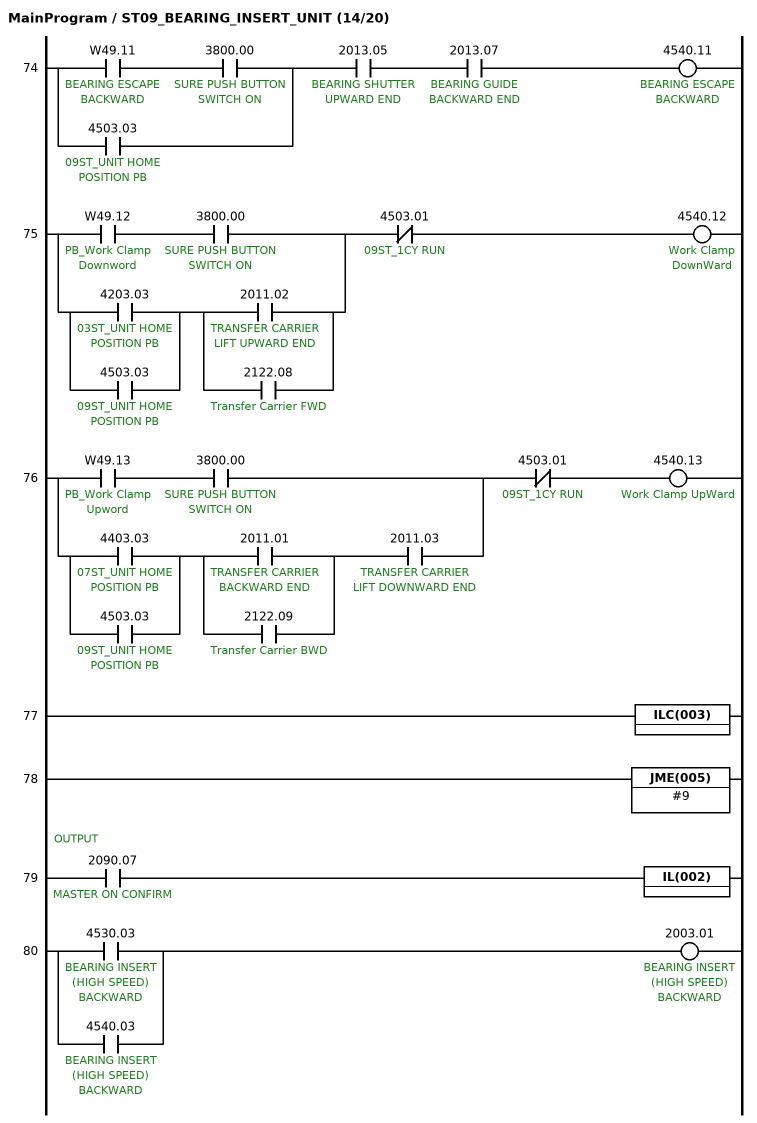
; [picture p480: MainProgram / ST09_BEARING_INSERT_UNIT, rungs 74-80]
; rung 74
LD W49.11  ; BEARING ESCAPE BACKWARD
AND 3800.00  ; SURE PUSH BUTTON SWITCH ON
OR 4503.03  ; 09ST_UNIT HOME POSITION PB
AND 2013.05  ; BEARING SHUTTER UPWARD END
AND 2013.07  ; BEARING GUIDE BACKWARD END
OUT 4540.11  ; BEARING ESCAPE BACKWARD
; rung 75
LD W49.12  ; PB_Work Clamp Downword
AND 3800.00  ; SURE PUSH BUTTON SWITCH ON
LD 4203.03  ; 03ST_UNIT HOME POSITION PB
OR 4503.03  ; 09ST_UNIT HOME POSITION PB
LD 2011.02  ; TRANSFER CARRIER LIFT UPWARD END
OR 2122.08  ; Transfer Carrier FWD
ANDLD
ORLD
ANDNOT 4503.01  ; 09ST_1CY RUN
OUT 4540.12  ; Work Clamp DownWard
; rung 76
LD W49.13  ; PB_Work Clamp Upword
AND 3800.00  ; SURE PUSH BUTTON SWITCH ON
LD 4403.03  ; 07ST_UNIT HOME POSITION PB
OR 4503.03  ; 09ST_UNIT HOME POSITION PB
LD 2011.01  ; TRANSFER CARRIER BACKWARD END
OR 2122.09  ; Transfer Carrier BWD
ANDLD
AND 2011.03  ; TRANSFER CARRIER LIFT DOWNWARD END
ORLD
ANDNOT 4503.01  ; 09ST_1CY RUN
OUT 4540.13  ; Work Clamp UpWard
; rung 77
ILC(003)
; rung 78
JME(005) #9
; rung 79: OUTPUT
LD 2090.07  ; MASTER ON CONFIRM
IL(002)
; rung 80
LD 4530.03  ; BEARING INSERT (HIGH SPEED) BACKWARD
OR 4540.03  ; BEARING INSERT (HIGH SPEED) BACKWARD
OUT 2003.01  ; BEARING INSERT (HIGH SPEED) BACKWARD

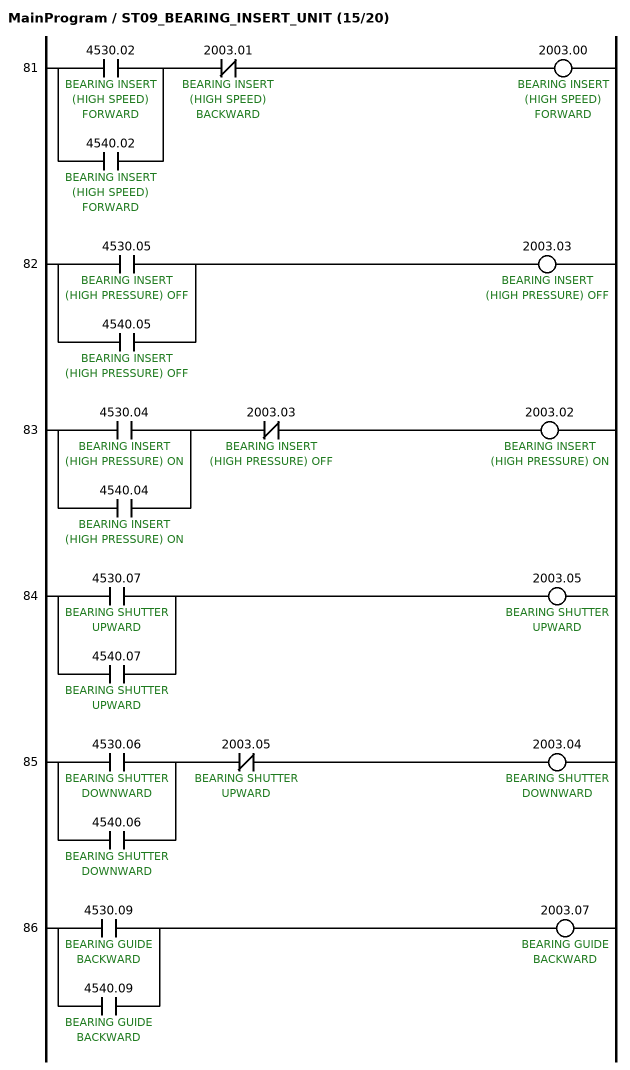
; rung 81
LD 4530.02  ; BEARING INSERT (HIGH SPEED) FORWARD
OR 4540.02  ; BEARING INSERT (HIGH SPEED) FORWARD
ANDNOT 2003.01  ; BEARING INSERT (HIGH SPEED) BACKWARD
OUT 2003.00  ; BEARING INSERT (HIGH SPEED) FORWARD
; rung 82
LD 4530.05  ; BEARING INSERT (HIGH PRESSURE) OFF
OR 4540.05  ; BEARING INSERT (HIGH PRESSURE) OFF
OUT 2003.03  ; BEARING INSERT (HIGH PRESSURE) OFF
; rung 83
LD 4530.04  ; BEARING INSERT (HIGH PRESSURE) ON
OR 4540.04  ; BEARING INSERT (HIGH PRESSURE) ON
ANDNOT 2003.03  ; BEARING INSERT (HIGH PRESSURE) OFF
OUT 2003.02  ; BEARING INSERT (HIGH PRESSURE) ON
; rung 84
LD 4530.07  ; BEARING SHUTTER UPWARD
OR 4540.07  ; BEARING SHUTTER UPWARD
OUT 2003.05  ; BEARING SHUTTER UPWARD
; rung 85
LD 4530.06  ; BEARING SHUTTER DOWNWARD
OR 4540.06  ; BEARING SHUTTER DOWNWARD
ANDNOT 2003.05  ; BEARING SHUTTER UPWARD
OUT 2003.04  ; BEARING SHUTTER DOWNWARD
; rung 86
LD 4530.09  ; BEARING GUIDE BACKWARD
OR 4540.09  ; BEARING GUIDE BACKWARD
OUT 2003.07  ; BEARING GUIDE BACKWARD

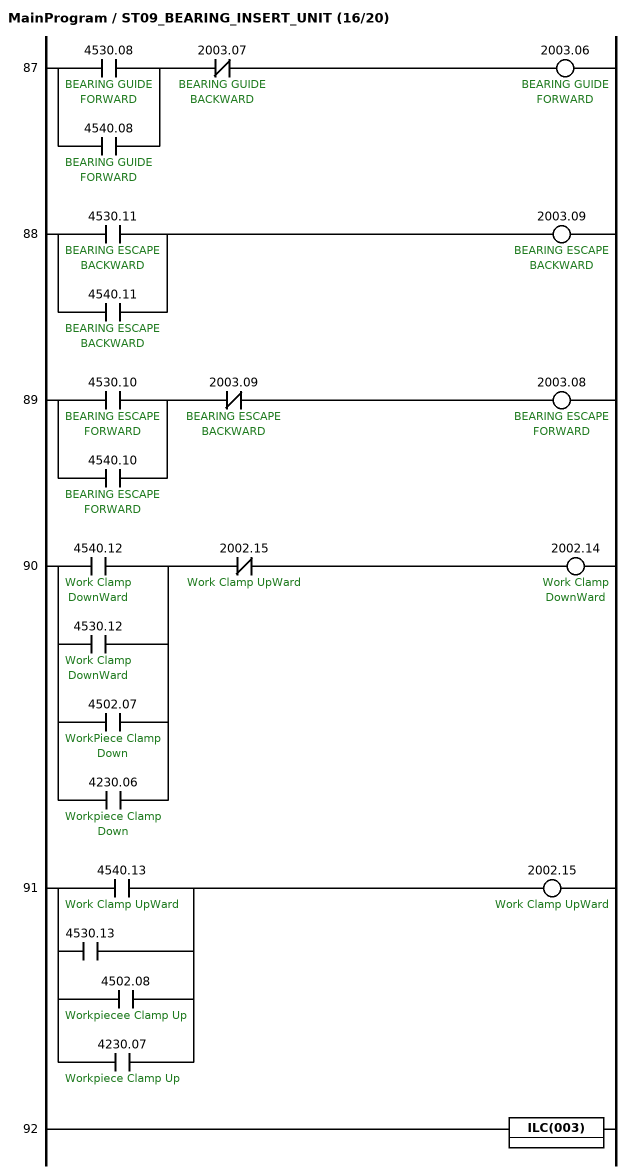
; rung 87
LD 4530.08  ; BEARING GUIDE FORWARD
OR 4540.08  ; BEARING GUIDE FORWARD
ANDNOT 2003.07  ; BEARING GUIDE BACKWARD
OUT 2003.06  ; BEARING GUIDE FORWARD
; rung 88
LD 4530.11  ; BEARING ESCAPE BACKWARD
OR 4540.11  ; BEARING ESCAPE BACKWARD
OUT 2003.09  ; BEARING ESCAPE BACKWARD
; rung 89
LD 4530.10  ; BEARING ESCAPE FORWARD
OR 4540.10  ; BEARING ESCAPE FORWARD
ANDNOT 2003.09  ; BEARING ESCAPE BACKWARD
OUT 2003.08  ; BEARING ESCAPE FORWARD
; rung 90
LD 4540.12  ; Work Clamp DownWard
OR 4530.12  ; Work Clamp DownWard
OR 4502.07  ; WorkPiece Clamp Down
OR 4230.06  ; Workpiece Clamp Down
ANDNOT 2002.15  ; Work Clamp UpWard
OUT 2002.14  ; Work Clamp DownWard
; rung 91
LD 4540.13  ; Work Clamp UpWard
OR 4530.13
OR 4502.08  ; Workpiecee Clamp Up
OR 4230.07  ; Workpiece Clamp Up
OUT 2002.15  ; Work Clamp UpWard
; rung 92
ILC(003)

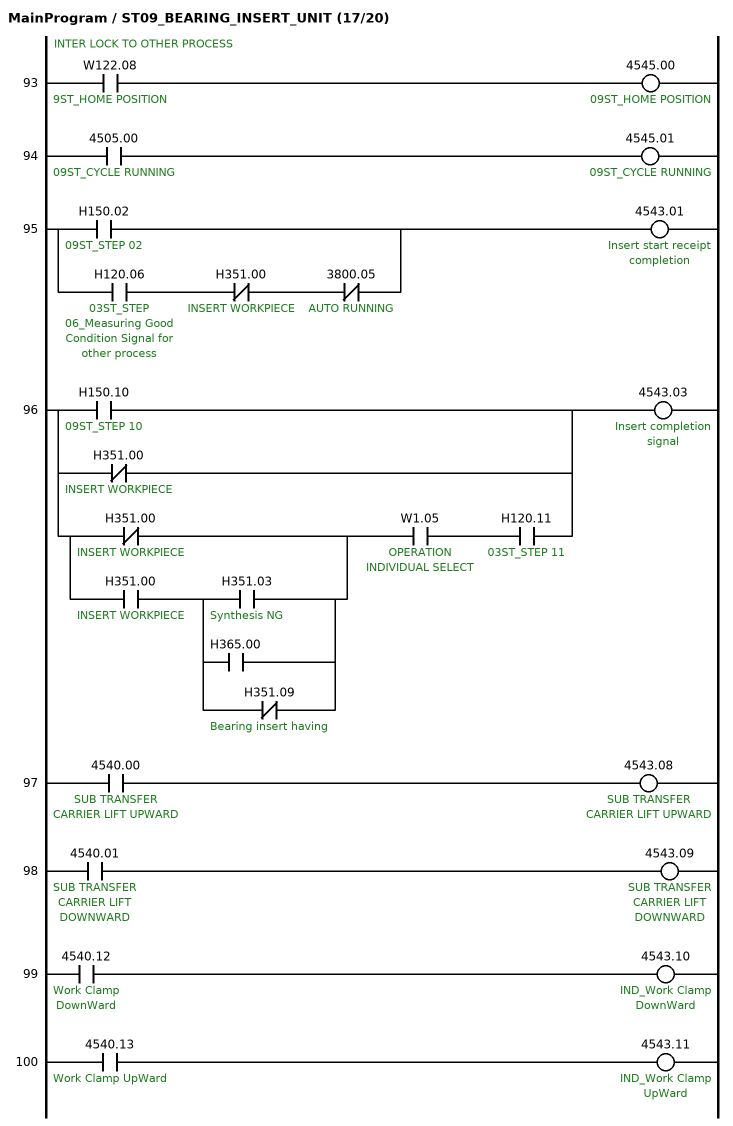
; rung 93: INTER LOCK TO OTHER PROCESS
LD W122.08  ; 9ST_HOME POSITION
OUT 4545.00  ; 09ST_HOME POSITION
; rung 94
LD 4505.00  ; 09ST_CYCLE RUNNING
OUT 4545.01  ; 09ST_CYCLE RUNNING
; rung 95
LD H150.02  ; 09ST_STEP 02
LD H120.06  ; 03ST_STEP 06_Measuring Good Condition Signal for other process
ANDNOT H351.00  ; INSERT WORKPIECE
ANDNOT 3800.05  ; AUTO RUNNING
ORLD
OUT 4543.01  ; Insert start receipt completion
; rung 96
LD H150.10  ; 09ST_STEP 10
ORNOT H351.00  ; INSERT WORKPIECE
LDNOT H351.00  ; INSERT WORKPIECE
LD H351.00  ; INSERT WORKPIECE
LD H351.03  ; Synthesis NG
OR H365.00
ORNOT H351.09  ; Bearing insert having
ANDLD
ORLD
AND W1.05  ; OPERATION INDIVIDUAL SELECT
AND H120.11  ; 03ST_STEP 11
ORLD
OUT 4543.03  ; Insert completion signal
; rung 97
LD 4540.00  ; SUB TRANSFER CARRIER LIFT UPWARD
OUT 4543.08  ; SUB TRANSFER CARRIER LIFT UPWARD
; rung 98
LD 4540.01  ; SUB TRANSFER CARRIER LIFT DOWNWARD
OUT 4543.09  ; SUB TRANSFER CARRIER LIFT DOWNWARD
; rung 99
LD 4540.12  ; Work Clamp DownWard
OUT 4543.10  ; IND_Work Clamp DownWard
; rung 100
LD 4540.13  ; Work Clamp UpWard
OUT 4543.11  ; IND_Work Clamp UpWard

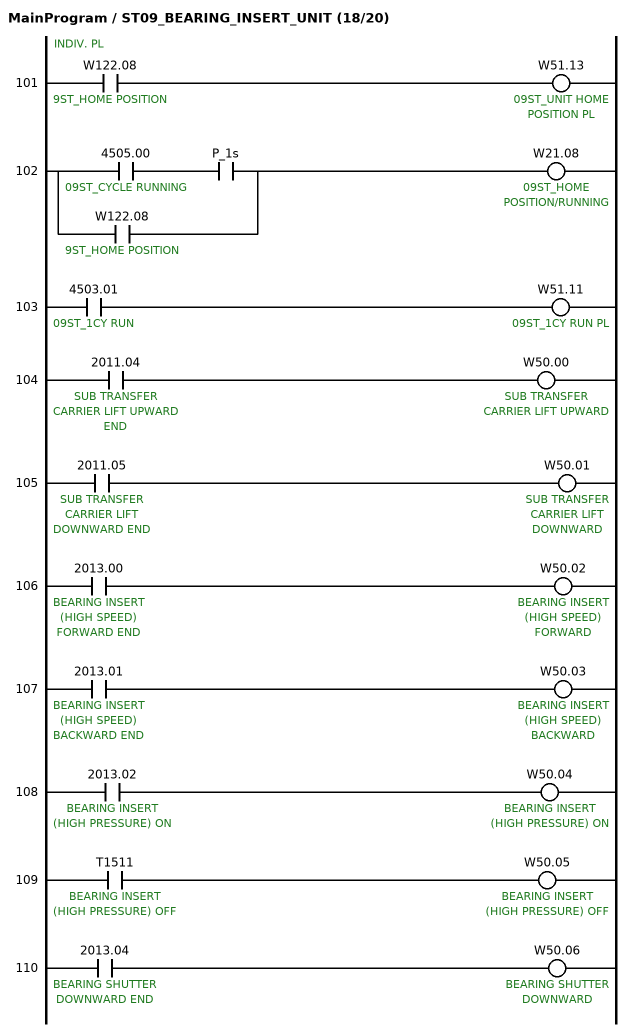
; rung 101: INDIV. PL
LD W122.08  ; 9ST_HOME POSITION
OUT W51.13  ; 09ST_UNIT HOME POSITION PL
; rung 102
LD 4505.00  ; 09ST_CYCLE RUNNING
AND P_1s
OR W122.08  ; 9ST_HOME POSITION
OUT W21.08  ; 09ST_HOME POSITION/RUNNING
; rung 103
LD 4503.01  ; 09ST_1CY RUN
OUT W51.11  ; 09ST_1CY RUN PL
; rung 104
LD 2011.04  ; SUB TRANSFER CARRIER LIFT UPWARD END
OUT W50.00  ; SUB TRANSFER CARRIER LIFT UPWARD
; rung 105
LD 2011.05  ; SUB TRANSFER CARRIER LIFT DOWNWARD END
OUT W50.01  ; SUB TRANSFER CARRIER LIFT DOWNWARD
; rung 106
LD 2013.00  ; BEARING INSERT (HIGH SPEED) FORWARD END
OUT W50.02  ; BEARING INSERT (HIGH SPEED) FORWARD
; rung 107
LD 2013.01  ; BEARING INSERT (HIGH SPEED) BACKWARD END
OUT W50.03  ; BEARING INSERT (HIGH SPEED) BACKWARD
; rung 108
LD 2013.02  ; BEARING INSERT (HIGH PRESSURE) ON
OUT W50.04  ; BEARING INSERT (HIGH PRESSURE) ON
; rung 109
LD T1511  ; BEARING INSERT (HIGH PRESSURE) OFF
OUT W50.05  ; BEARING INSERT (HIGH PRESSURE) OFF
; rung 110
LD 2013.04  ; BEARING SHUTTER DOWNWARD END
OUT W50.06  ; BEARING SHUTTER DOWNWARD

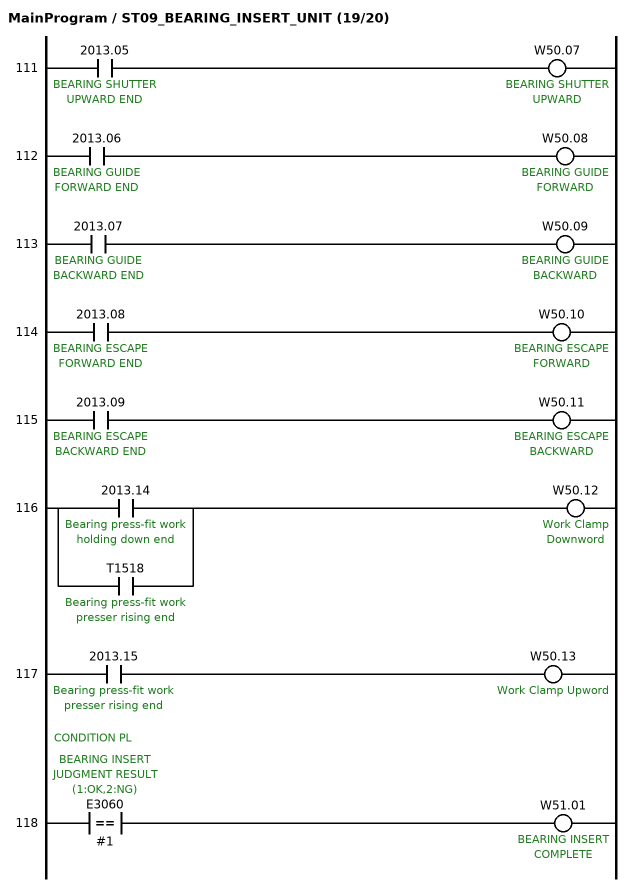
; rung 111
LD 2013.05  ; BEARING SHUTTER UPWARD END
OUT W50.07  ; BEARING SHUTTER UPWARD
; rung 112
LD 2013.06  ; BEARING GUIDE FORWARD END
OUT W50.08  ; BEARING GUIDE FORWARD
; rung 113
LD 2013.07  ; BEARING GUIDE BACKWARD END
OUT W50.09  ; BEARING GUIDE BACKWARD
; rung 114
LD 2013.08  ; BEARING ESCAPE FORWARD END
OUT W50.10  ; BEARING ESCAPE FORWARD
; rung 115
LD 2013.09  ; BEARING ESCAPE BACKWARD END
OUT W50.11  ; BEARING ESCAPE BACKWARD
; rung 116
LD 2013.14  ; Bearing press-fit work holding down end
OR T1518  ; Bearing press-fit work presser rising end
OUT W50.12  ; Work Clamp Downword
; rung 117
LD 2013.15  ; Bearing press-fit work presser rising end
OUT W50.13  ; Work Clamp Upword
; rung 118: CONDITION PL
LD=(300) E3060 #1  ; BEARING INSERT JUDGMENT RESULT (1:OK,2:NG)
OUT W51.01  ; BEARING INSERT COMPLETE

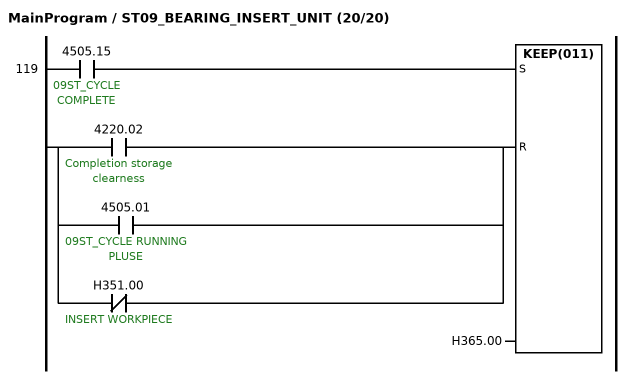
; rung 119
LD 4505.15  ; 09ST_CYCLE COMPLETE
LD 4220.02  ; Completion storage clearness
OR 4505.01  ; 09ST_CYCLE RUNNING PLUSE
ORNOT H351.00  ; INSERT WORKPIECE
KEEP(011) H365.00

### Section ST10_LENGTH_MEASURE_UNIT

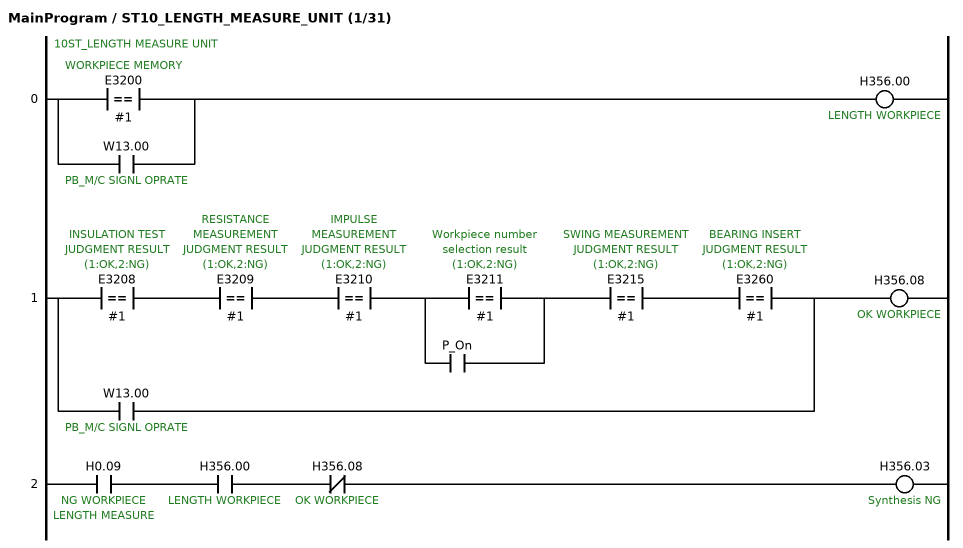
; rung 0: 10ST_LENGTH MEASURE UNIT
LD=(300) E3200 #1  ; WORKPIECE MEMORY
OR W13.00  ; PB_M/C SIGNL OPRATE
OUT H356.00  ; LENGTH WORKPIECE
; rung 1
LD=(300) E3208 #1  ; INSULATION TEST JUDGMENT RESULT (1:OK,2:NG)
AND=(300) E3209 #1  ; RESISTANCE MEASUREMENT JUDGMENT RESULT (1:OK,2:NG)
AND=(300) E3210 #1  ; IMPULSE MEASUREMENT JUDGMENT RESULT (1:OK,2:NG)
LD=(300) E3211 #1  ; Workpiece number selection result (1:OK,2:NG)
OR P_On
ANDLD
AND=(300) E3215 #1  ; SWING MEASUREMENT JUDGMENT RESULT (1:OK,2:NG)
AND=(300) E3260 #1  ; BEARING INSERT JUDGMENT RESULT (1:OK,2:NG)
OR W13.00  ; PB_M/C SIGNL OPRATE
OUT H356.08  ; OK WORKPIECE
; rung 2
LD H0.09  ; NG WORKPIECE LENGTH MEASURE
AND H356.00  ; LENGTH WORKPIECE
ANDNOT H356.08  ; OK WORKPIECE
OUT H356.03  ; Synthesis NG

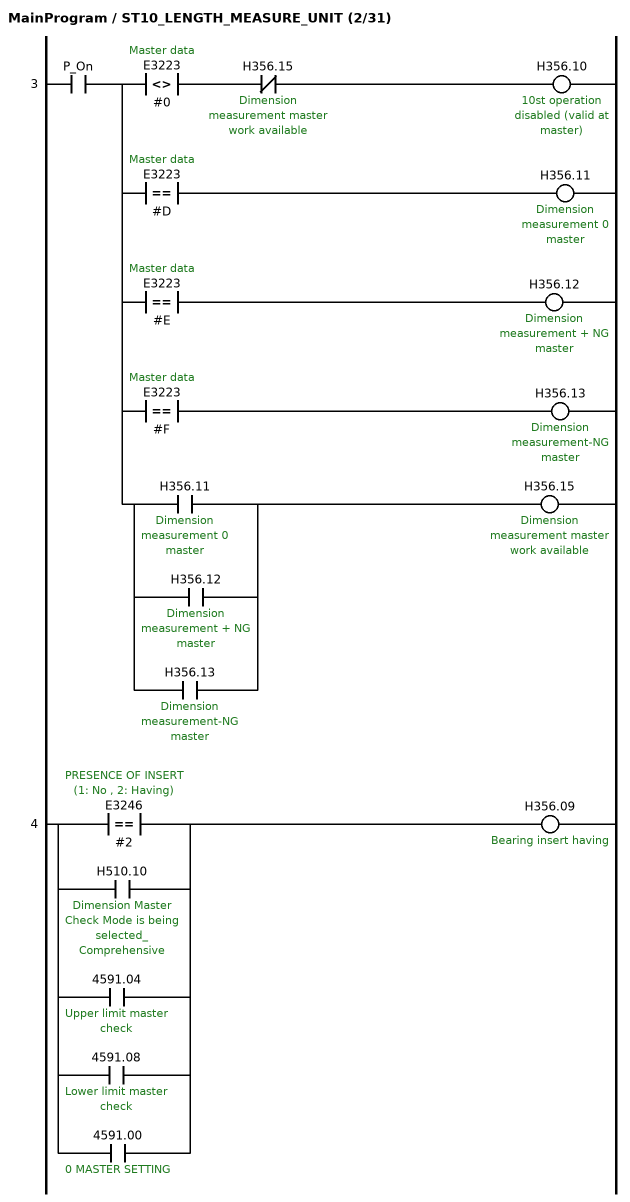
; rung 3
LD P_On
OUT TR0
AND<>(305) E3223 #0  ; Master data
ANDNOT H356.15  ; Dimension measurement master work available
OUT H356.10  ; 10st operation disabled (valid at master)
LD TR0
AND=(300) E3223 #D  ; Master data
OUT H356.11  ; Dimension measurement 0 master
LD TR0
AND=(300) E3223 #E  ; Master data
OUT H356.12  ; Dimension measurement + NG master
LD TR0
AND=(300) E3223 #F  ; Master data
OUT H356.13  ; Dimension measurement-NG master
LD TR0
LD H356.11  ; Dimension measurement 0 master
OR H356.12  ; Dimension measurement + NG master
OR H356.13  ; Dimension measurement-NG master
ANDLD
OUT H356.15  ; Dimension measurement master work available
; rung 4
LD=(300) E3246 #2  ; PRESENCE OF INSERT (1: No , 2: Having)
OR H510.10  ; Dimension Master Check Mode is being selected_Comprehensive
OR 4591.04  ; Upper limit master check
OR 4591.08  ; Lower limit master check
OR 4591.00  ; 0 MASTER SETTING
OUT H356.09  ; Bearing insert having

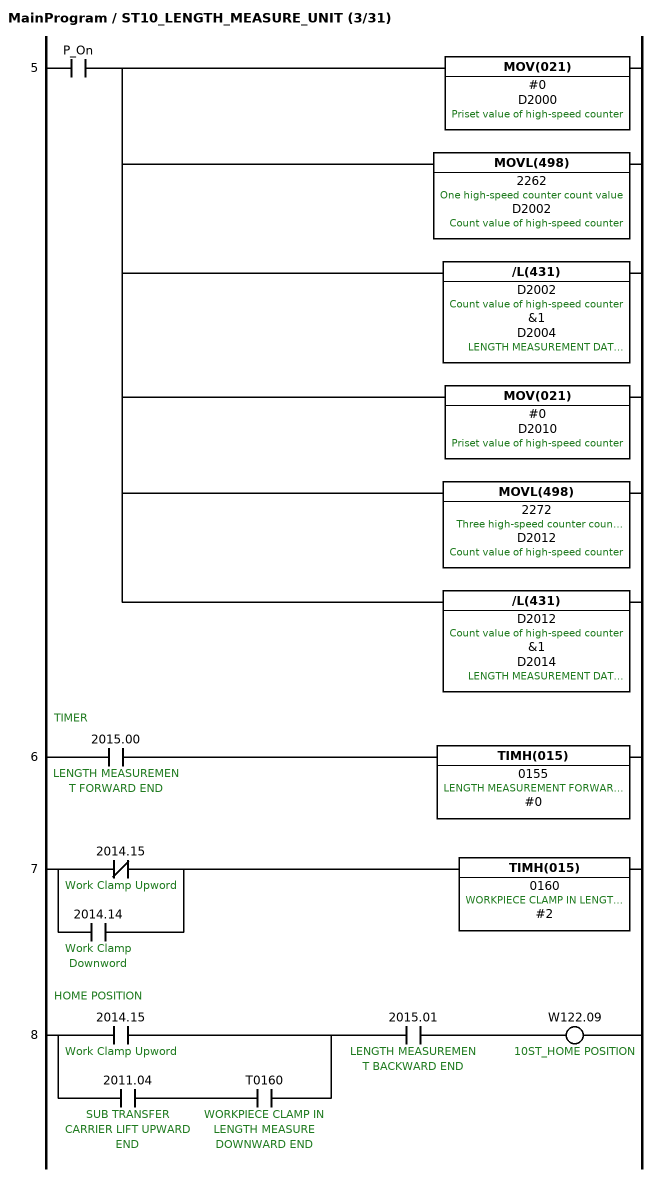
; rung 5
LD P_On
MOV(021) #0 D2000  ; Priset value of high-speed counter
MOVL(498) 2262 D2002  ; One high-speed counter count value, Count value of high-speed counter
/L(431) D2002 &1 D2004  ; Count value of high-speed counter, LENGTH MEASUREMENT DATA (OVERALL)
MOV(021) #0 D2010  ; Priset value of high-speed counter
MOVL(498) 2272 D2012  ; Three high-speed counter count value, Count value of high-speed counter
/L(431) D2012 &1 D2014  ; Count value of high-speed counter, LENGTH MEASUREMENT DATA (BEARING)
; rung 6: TIMER
LD 2015.00  ; LENGTH MEASUREMENT FORWARD END
TIMH(015) 0155 #0  ; LENGTH MEASUREMENT FORWARD END
; rung 7
LDNOT 2014.15  ; Work Clamp Upword
OR 2014.14  ; Work Clamp Downword
TIMH(015) 0160 #2  ; WORKPIECE CLAMP IN LENGTH MEASURE DOWNWARD END
; rung 8: HOME POSITION
LD 2014.15  ; Work Clamp Upword
LD 2011.04  ; SUB TRANSFER CARRIER LIFT UPWARD END
AND T0160  ; WORKPIECE CLAMP IN LENGTH MEASURE DOWNWARD END
ORLD
AND 2015.01  ; LENGTH MEASUREMENT BACKWARD END
OUT W122.09  ; 10ST_HOME POSITION

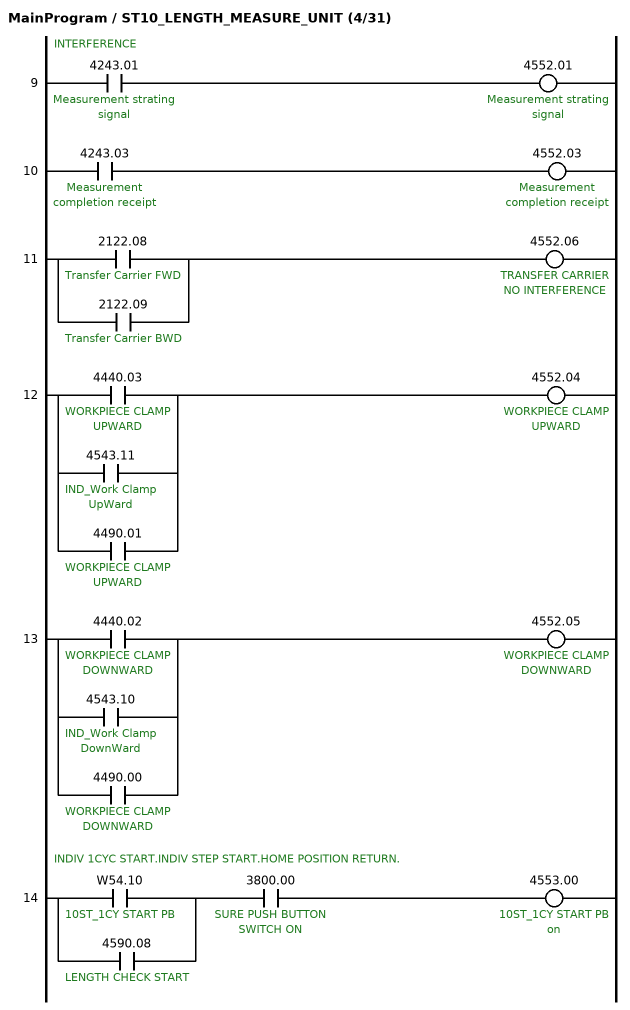
; rung 9: INTERFERENCE
LD 4243.01  ; Measurement strating signal
OUT 4552.01  ; Measurement strating signal
; rung 10
LD 4243.03  ; Measurement completion receipt
OUT 4552.03  ; Measurement completion receipt
; rung 11
LD 2122.08  ; Transfer Carrier FWD
OR 2122.09  ; Transfer Carrier BWD
OUT 4552.06  ; TRANSFER CARRIER NO INTERFERENCE
; rung 12
LD 4440.03  ; WORKPIECE CLAMP UPWARD
OR 4543.11  ; IND_Work Clamp UpWard
OR 4490.01  ; WORKPIECE CLAMP UPWARD
OUT 4552.04  ; WORKPIECE CLAMP UPWARD
; rung 13
LD 4440.02  ; WORKPIECE CLAMP DOWNWARD
OR 4543.10  ; IND_Work Clamp DownWard
OR 4490.00  ; WORKPIECE CLAMP DOWNWARD
OUT 4552.05  ; WORKPIECE CLAMP DOWNWARD
; rung 14: INDIV 1CYC START.INDIV STEP START.HOME POSITION RETURN.
LD W54.10  ; 10ST_1CY START PB
OR 4590.08  ; LENGTH CHECK START
AND 3800.00  ; SURE PUSH BUTTON SWITCH ON
OUT 4553.00  ; 10ST_1CY START PB on

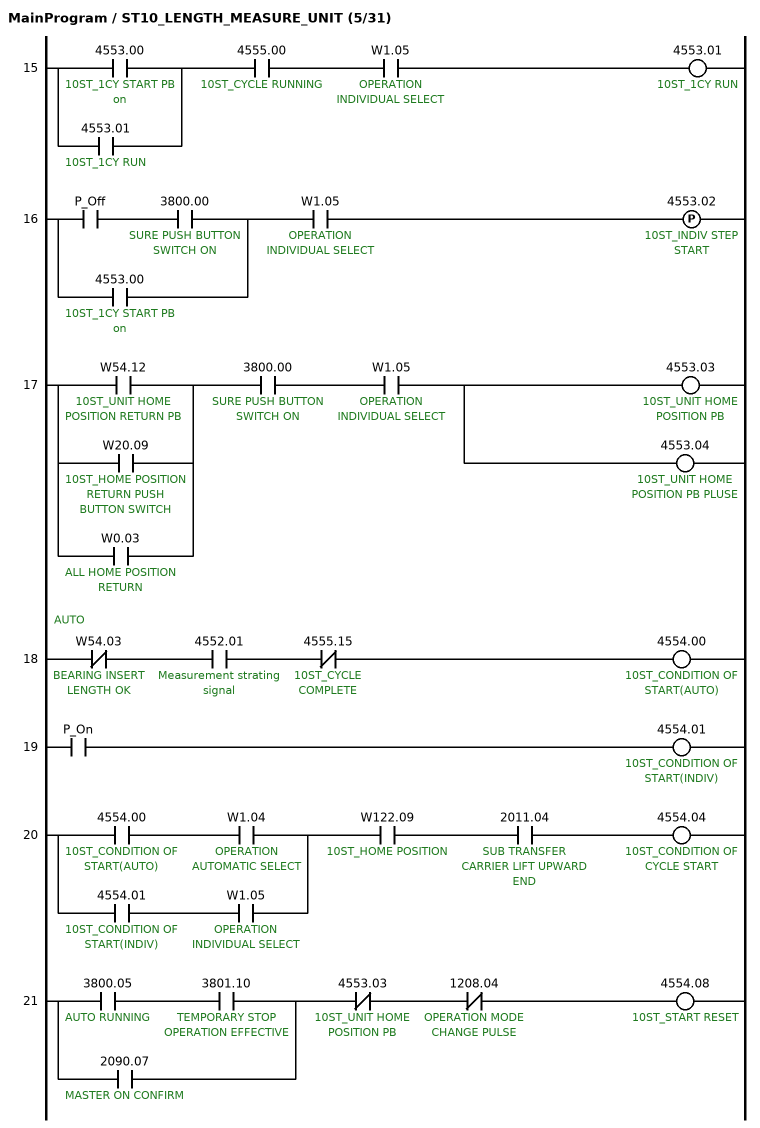
; rung 15
LD 4553.00  ; 10ST_1CY START PB on
OR 4553.01  ; 10ST_1CY RUN
AND 4555.00  ; 10ST_CYCLE RUNNING
AND W1.05  ; OPERATION INDIVIDUAL SELECT
OUT 4553.01  ; 10ST_1CY RUN
; rung 16
LD P_Off
AND 3800.00  ; SURE PUSH BUTTON SWITCH ON
OR 4553.00  ; 10ST_1CY START PB on
AND W1.05  ; OPERATION INDIVIDUAL SELECT
DIFU(013) 4553.02  ; 10ST_INDIV STEP START
; rung 17
LD W54.12  ; 10ST_UNIT HOME POSITION RETURN PB
OR W20.09  ; 10ST_HOME POSITION RETURN PUSH BUTTON SWITCH
OR W0.03  ; ALL HOME POSITION RETURN
AND 3800.00  ; SURE PUSH BUTTON SWITCH ON
AND W1.05  ; OPERATION INDIVIDUAL SELECT
OUT 4553.03  ; 10ST_UNIT HOME POSITION PB
OUT 4553.04  ; 10ST_UNIT HOME POSITION PB PLUSE
; rung 18: AUTO
LDNOT W54.03  ; BEARING INSERT LENGTH OK
AND 4552.01  ; Measurement strating signal
ANDNOT 4555.15  ; 10ST_CYCLE COMPLETE
OUT 4554.00  ; 10ST_CONDITION OF START(AUTO)
; rung 19
LD P_On
OUT 4554.01  ; 10ST_CONDITION OF START(INDIV)
; rung 20
LD 4554.00  ; 10ST_CONDITION OF START(AUTO)
AND W1.04  ; OPERATION AUTOMATIC SELECT
LD 4554.01  ; 10ST_CONDITION OF START(INDIV)
AND W1.05  ; OPERATION INDIVIDUAL SELECT
ORLD
AND W122.09  ; 10ST_HOME POSITION
AND 2011.04  ; SUB TRANSFER CARRIER LIFT UPWARD END
OUT 4554.04  ; 10ST_CONDITION OF CYCLE START
; rung 21
LD 3800.05  ; AUTO RUNNING
AND 3801.10  ; TEMPORARY STOP OPERATION EFFECTIVE
OR 2090.07  ; MASTER ON CONFIRM
ANDNOT 4553.03  ; 10ST_UNIT HOME POSITION PB
ANDNOT 1208.04  ; OPERATION MODE CHANGE PULSE
OUT 4554.08  ; 10ST_START RESET

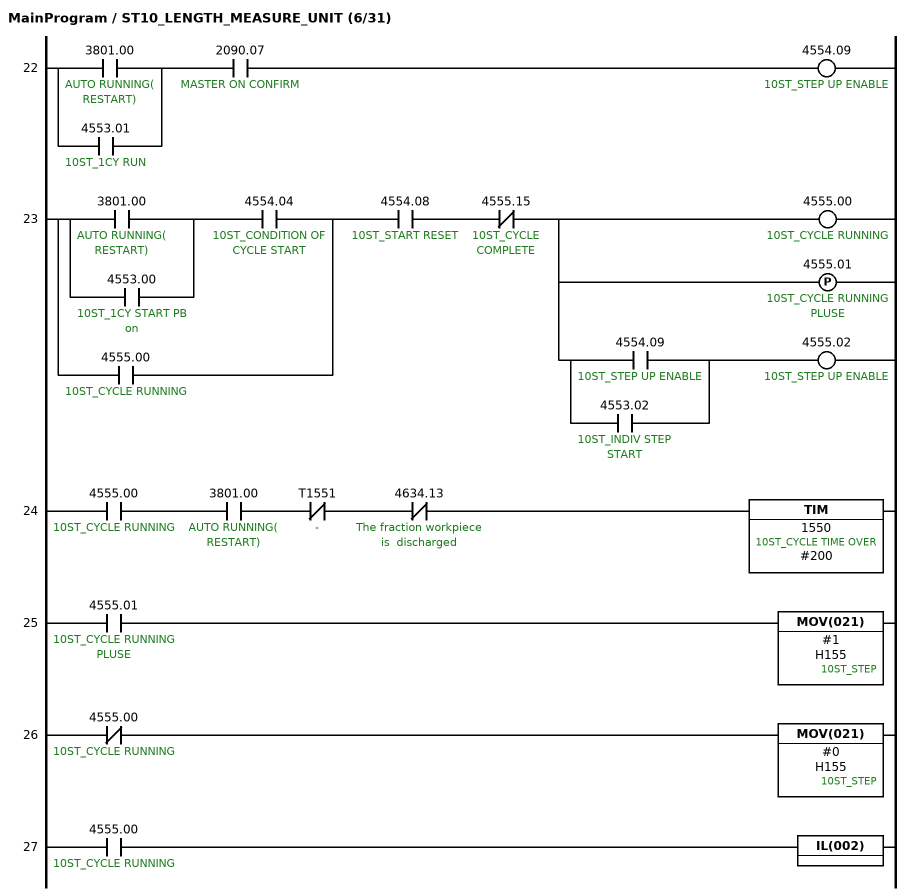
; rung 22
LD 3801.00  ; AUTO RUNNING(RESTART)
OR 4553.01  ; 10ST_1CY RUN
AND 2090.07  ; MASTER ON CONFIRM
OUT 4554.09  ; 10ST_STEP UP ENABLE
; rung 23
LD 3801.00  ; AUTO RUNNING(RESTART)
OR 4553.00  ; 10ST_1CY START PB on
AND 4554.04  ; 10ST_CONDITION OF CYCLE START
OR 4555.00  ; 10ST_CYCLE RUNNING
AND 4554.08  ; 10ST_START RESET
ANDNOT 4555.15  ; 10ST_CYCLE COMPLETE
OUT 4555.00  ; 10ST_CYCLE RUNNING
DIFU(013) 4555.01  ; 10ST_CYCLE RUNNING PLUSE
LD 4554.09  ; 10ST_STEP UP ENABLE
OR 4553.02  ; 10ST_INDIV STEP START
ANDLD
OUT 4555.02  ; 10ST_STEP UP ENABLE
; rung 24
LD 4555.00  ; 10ST_CYCLE RUNNING
AND 3801.00  ; AUTO RUNNING(RESTART)
ANDNOT T1551  ; -
ANDNOT 4634.13  ; The fraction workpiece is  discharged
TIM 1550 #200  ; 10ST_CYCLE TIME OVER
; rung 25
LD 4555.01  ; 10ST_CYCLE RUNNING PLUSE
MOV(021) #1 H155  ; 10ST_STEP
; rung 26
LDNOT 4555.00  ; 10ST_CYCLE RUNNING
MOV(021) #0 H155  ; 10ST_STEP
; rung 27
LD 4555.00  ; 10ST_CYCLE RUNNING
IL(002)

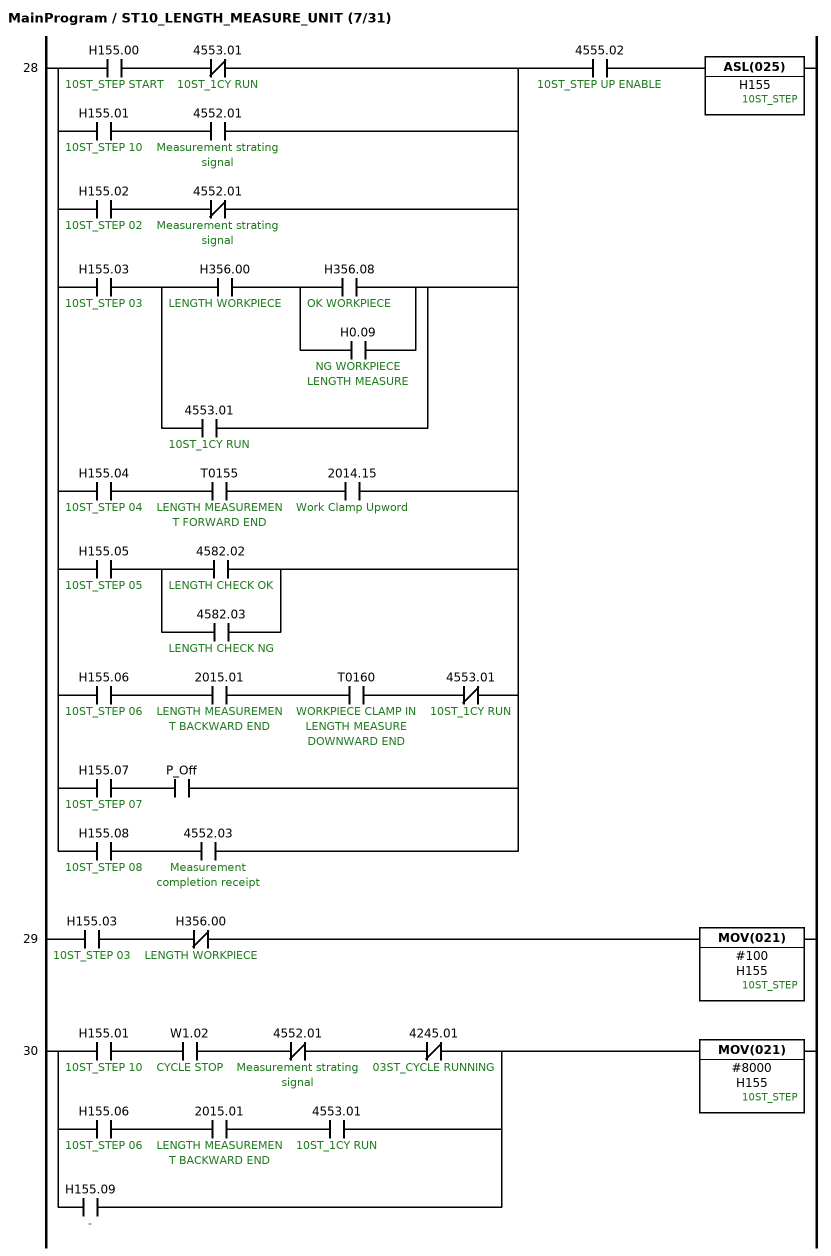
; rung 28
LD H155.00  ; 10ST_STEP START
ANDNOT 4553.01  ; 10ST_1CY RUN
LD H155.01  ; 10ST_STEP 10
AND 4552.01  ; Measurement strating signal
ORLD
LD H155.02  ; 10ST_STEP 02
ANDNOT 4552.01  ; Measurement strating signal
ORLD
LD H155.03  ; 10ST_STEP 03
LD H356.00  ; LENGTH WORKPIECE
LD H356.08  ; OK WORKPIECE
OR H0.09  ; NG WORKPIECE LENGTH MEASURE
ANDLD
OR 4553.01  ; 10ST_1CY RUN
ANDLD
ORLD
LD H155.04  ; 10ST_STEP 04
AND T0155  ; LENGTH MEASUREMENT FORWARD END
AND 2014.15  ; Work Clamp Upword
ORLD
LD H155.05  ; 10ST_STEP 05
LD 4582.02  ; LENGTH CHECK OK
OR 4582.03  ; LENGTH CHECK NG
ANDLD
ORLD
LD H155.06  ; 10ST_STEP 06
AND 2015.01  ; LENGTH MEASUREMENT BACKWARD END
AND T0160  ; WORKPIECE CLAMP IN LENGTH MEASURE DOWNWARD END
ANDNOT 4553.01  ; 10ST_1CY RUN
ORLD
LD H155.07  ; 10ST_STEP 07
AND P_Off
ORLD
LD H155.08  ; 10ST_STEP 08
AND 4552.03  ; Measurement completion receipt
ORLD
AND 4555.02  ; 10ST_STEP UP ENABLE
ASL(025) H155  ; 10ST_STEP
; rung 29
LD H155.03  ; 10ST_STEP 03
ANDNOT H356.00  ; LENGTH WORKPIECE
MOV(021) #100 H155  ; 10ST_STEP
; rung 30
LD H155.01  ; 10ST_STEP 10
AND W1.02  ; CYCLE STOP
ANDNOT 4552.01  ; Measurement strating signal
ANDNOT 4245.01  ; 03ST_CYCLE RUNNING
LD H155.06  ; 10ST_STEP 06
AND 2015.01  ; LENGTH MEASUREMENT BACKWARD END
AND 4553.01  ; 10ST_1CY RUN
ORLD
OR H155.09  ; -
MOV(021) #8000 H155  ; 10ST_STEP

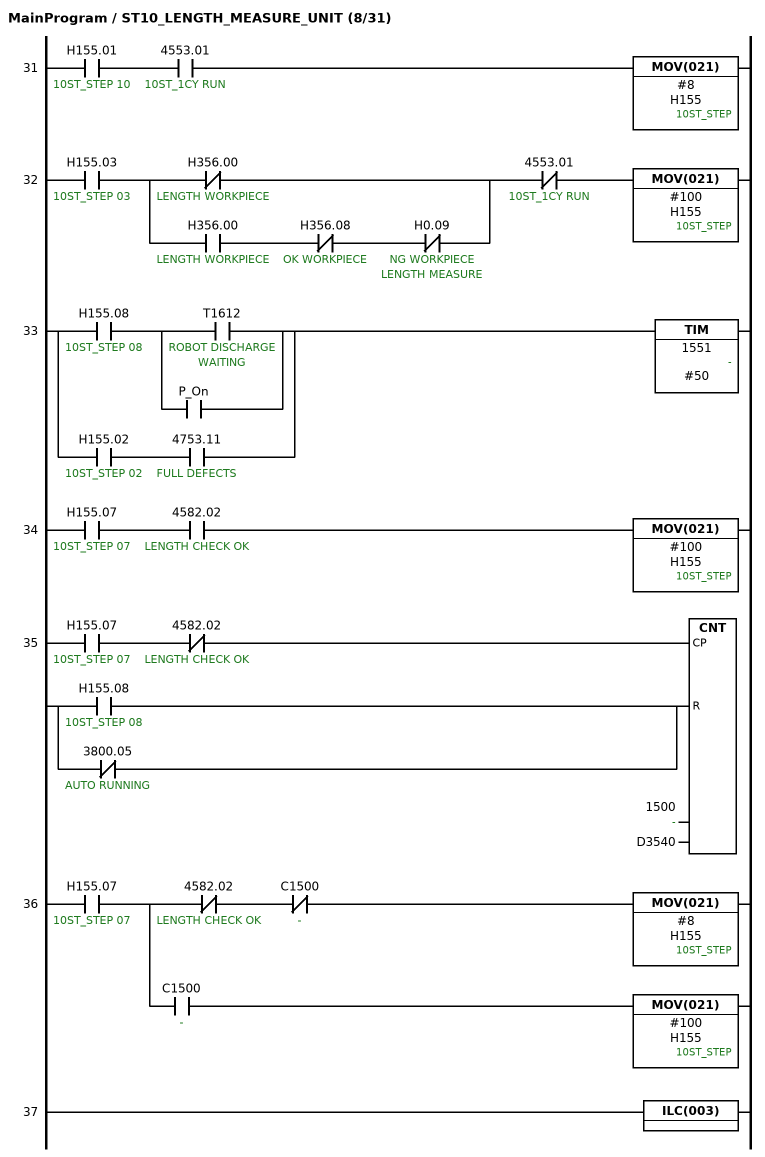
; rung 31
LD H155.01  ; 10ST_STEP 10
AND 4553.01  ; 10ST_1CY RUN
MOV(021) #8 H155  ; 10ST_STEP
; rung 32
LD H155.03  ; 10ST_STEP 03
LDNOT H356.00  ; LENGTH WORKPIECE
LD H356.00  ; LENGTH WORKPIECE
ANDNOT H356.08  ; OK WORKPIECE
ANDNOT H0.09  ; NG WORKPIECE LENGTH MEASURE
ORLD
ANDLD
ANDNOT 4553.01  ; 10ST_1CY RUN
MOV(021) #100 H155  ; 10ST_STEP
; rung 33
LD H155.08  ; 10ST_STEP 08
LD T1612  ; ROBOT DISCHARGE WAITING
OR P_On
ANDLD
LD H155.02  ; 10ST_STEP 02
AND 4753.11  ; FULL DEFECTS
ORLD
TIM 1551 #50  ; -
; rung 34
LD H155.07  ; 10ST_STEP 07
AND 4582.02  ; LENGTH CHECK OK
MOV(021) #100 H155  ; 10ST_STEP
; rung 35
LD H155.07  ; 10ST_STEP 07
ANDNOT 4582.02  ; LENGTH CHECK OK
LD H155.08  ; 10ST_STEP 08
ORNOT 3800.05  ; AUTO RUNNING
CNT 1500 D3540  ; -
; rung 36
LD H155.07  ; 10ST_STEP 07
OUT TR0
ANDNOT 4582.02  ; LENGTH CHECK OK
ANDNOT C1500  ; -
MOV(021) #8 H155  ; 10ST_STEP
LD TR0
AND C1500  ; -
MOV(021) #100 H155  ; 10ST_STEP
; rung 37
ILC(003)

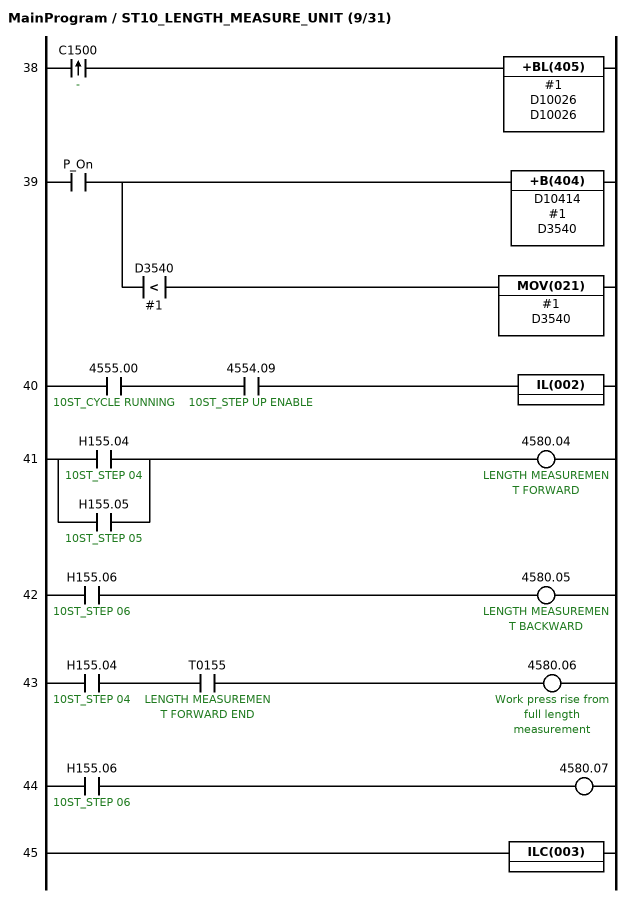
; rung 38
@LD C1500  ; -
+BL(405) #1 D10026 D10026
; rung 39
LD P_On
+B(404) D10414 #1 D3540
AND<(310) D3540 #1
MOV(021) #1 D3540
; rung 40
LD 4555.00  ; 10ST_CYCLE RUNNING
AND 4554.09  ; 10ST_STEP UP ENABLE
IL(002)
; rung 41
LD H155.04  ; 10ST_STEP 04
OR H155.05  ; 10ST_STEP 05
OUT 4580.04  ; LENGTH MEASUREMENT FORWARD
; rung 42
LD H155.06  ; 10ST_STEP 06
OUT 4580.05  ; LENGTH MEASUREMENT BACKWARD
; rung 43
LD H155.04  ; 10ST_STEP 04
AND T0155  ; LENGTH MEASUREMENT FORWARD END
OUT 4580.06  ; Work press rise from full length measurement
; rung 44
LD H155.06  ; 10ST_STEP 06
OUT 4580.07
; rung 45
ILC(003)

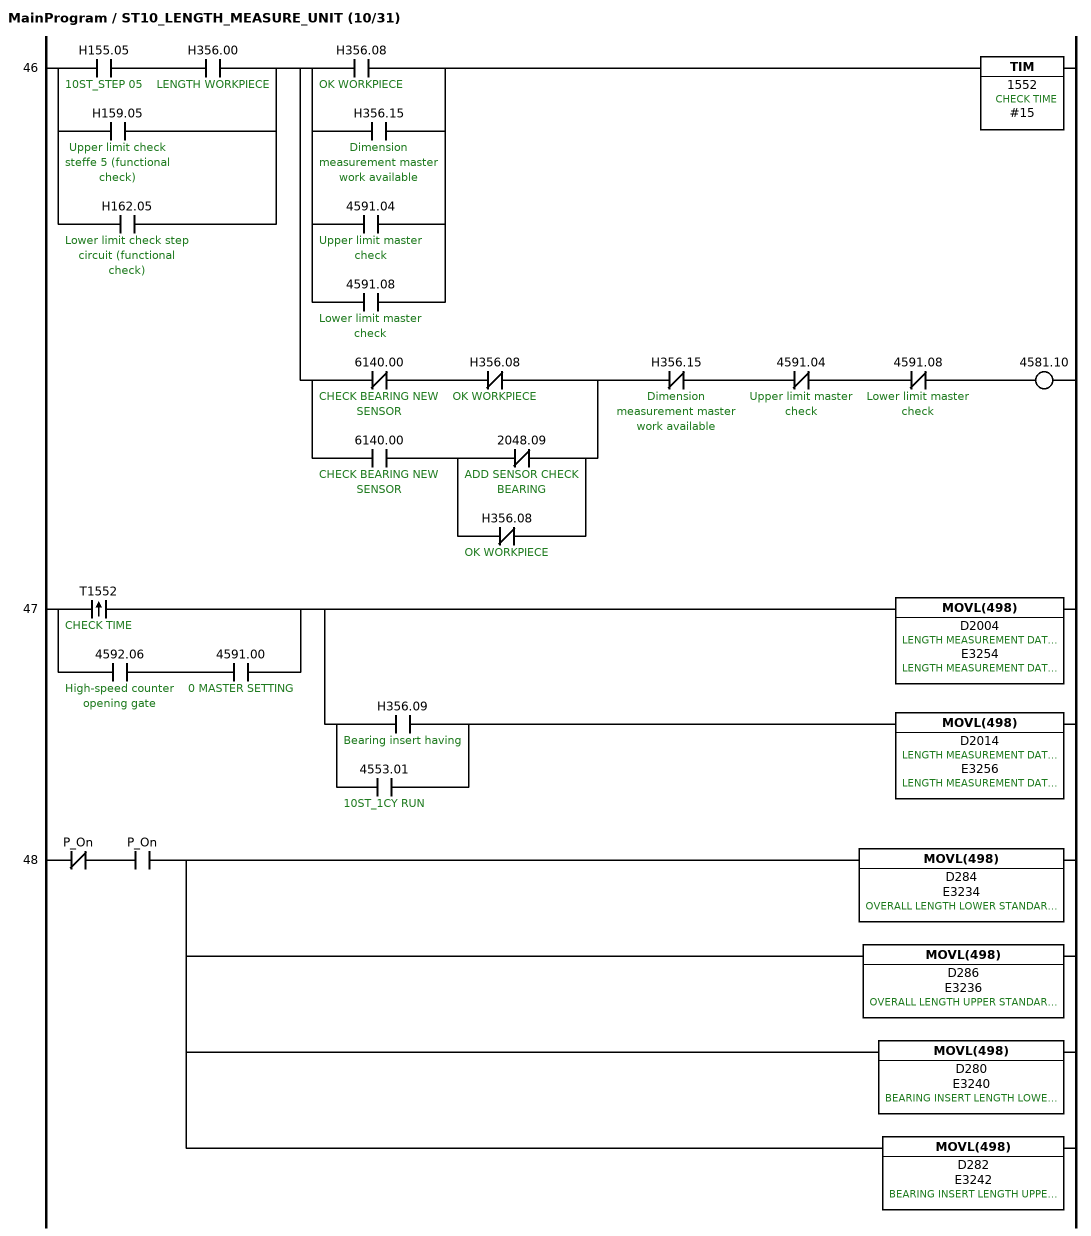
; rung 46
LD H155.05  ; 10ST_STEP 05
AND H356.00  ; LENGTH WORKPIECE
OR H159.05  ; Upper limit check steffe 5 (functional check)
OR H162.05  ; Lower limit check step circuit (functional check)
OUT TR0
LD H356.08  ; OK WORKPIECE
OR H356.15  ; Dimension measurement master work available
OR 4591.04  ; Upper limit master check
OR 4591.08  ; Lower limit master check
ANDLD
TIM 1552 #15  ; CHECK TIME
LD TR0
LDNOT 6140.00  ; CHECK BEARING NEW SENSOR
ANDNOT H356.08  ; OK WORKPIECE
LD 6140.00  ; CHECK BEARING NEW SENSOR
LDNOT 2048.09  ; ADD SENSOR CHECK BEARING
ORNOT H356.08  ; OK WORKPIECE
ANDLD
ORLD
ANDLD
ANDNOT H356.15  ; Dimension measurement master work available
ANDNOT 4591.04  ; Upper limit master check
ANDNOT 4591.08  ; Lower limit master check
OUT 4581.10
; rung 47
@LD T1552  ; CHECK TIME
LD 4592.06  ; High-speed counter opening gate
AND 4591.00  ; 0 MASTER SETTING
ORLD
MOVL(498) D2004 E3254  ; LENGTH MEASUREMENT DATA (OVERALL)
LD H356.09  ; Bearing insert having
OR 4553.01  ; 10ST_1CY RUN
ANDLD
MOVL(498) D2014 E3256  ; LENGTH MEASUREMENT DATA (BEARING)
; rung 48
LDNOT P_On
AND P_On
MOVL(498) D284 E3234  ; OVERALL LENGTH LOWER STANDARD VALUE
MOVL(498) D286 E3236  ; OVERALL LENGTH UPPER STANDARD VALUE
MOVL(498) D280 E3240  ; BEARING INSERT LENGTH LOWER STANDARD VALUE
MOVL(498) D282 E3242  ; BEARING INSERT LENGTH UPPER STANDARD VALUE

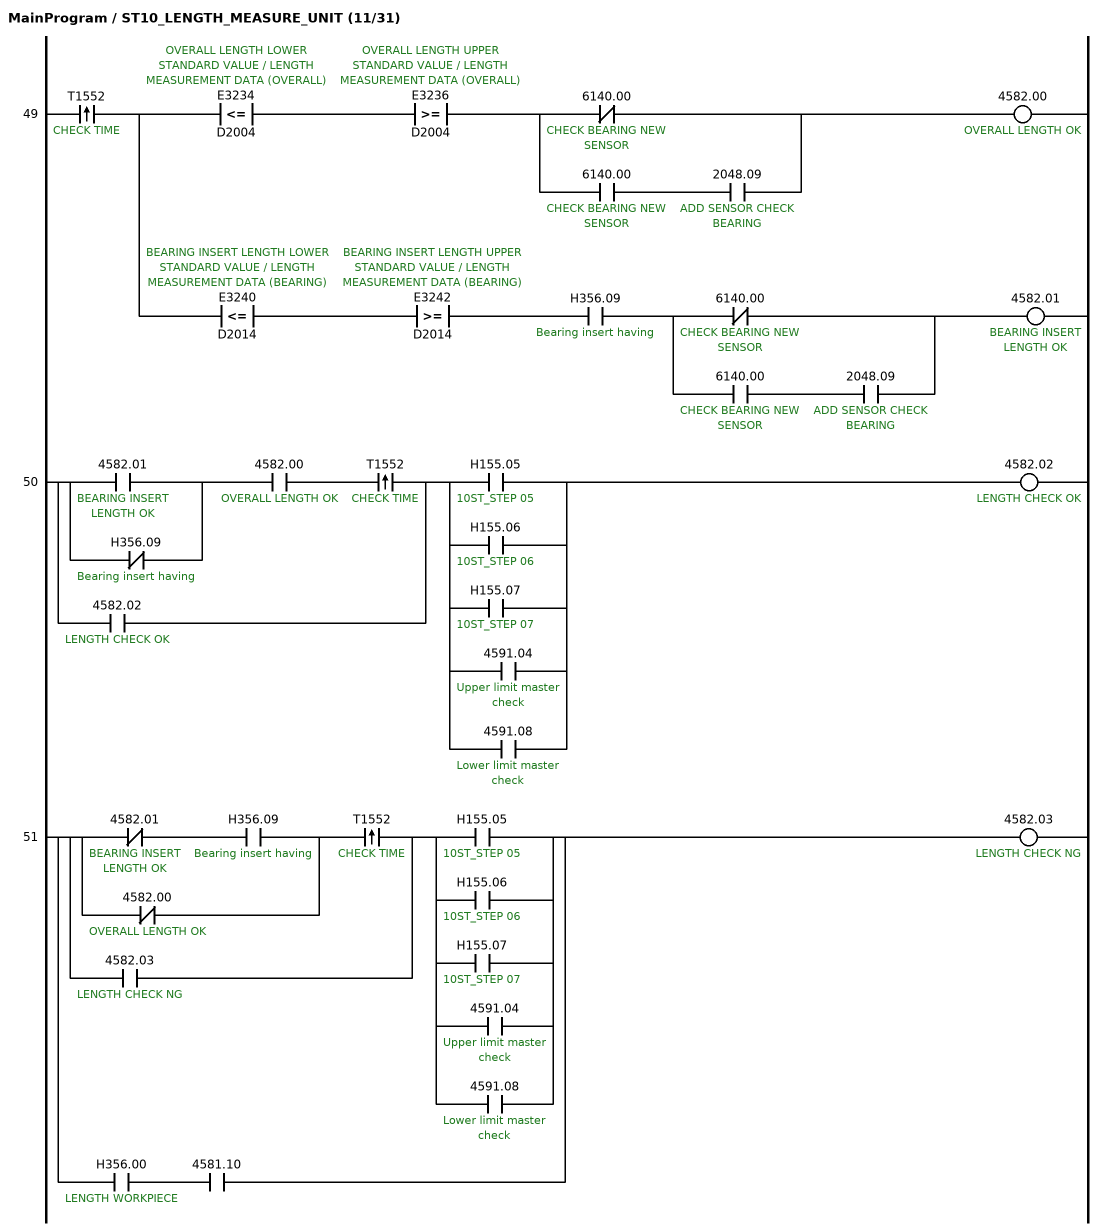
; rung 49
@LD T1552  ; CHECK TIME
OUT TR0
AND<=SL(318) E3234 D2004  ; OVERALL LENGTH LOWER STANDARD VALUE, LENGTH MEASUREMENT DATA (OVERALL)
AND>=SL(328) E3236 D2004  ; OVERALL LENGTH UPPER STANDARD VALUE, LENGTH MEASUREMENT DATA (OVERALL)
LDNOT 6140.00  ; CHECK BEARING NEW SENSOR
LD 6140.00  ; CHECK BEARING NEW SENSOR
AND 2048.09  ; ADD SENSOR CHECK BEARING
ORLD
ANDLD
OUT 4582.00  ; OVERALL LENGTH OK
LD TR0
AND<=SL(318) E3240 D2014  ; BEARING INSERT LENGTH LOWER STANDARD VALUE, LENGTH MEASUREMENT DATA (BEARING)
AND>=SL(328) E3242 D2014  ; BEARING INSERT LENGTH UPPER STANDARD VALUE, LENGTH MEASUREMENT DATA (BEARING)
AND H356.09  ; Bearing insert having
LDNOT 6140.00  ; CHECK BEARING NEW SENSOR
LD 6140.00  ; CHECK BEARING NEW SENSOR
AND 2048.09  ; ADD SENSOR CHECK BEARING
ORLD
ANDLD
OUT 4582.01  ; BEARING INSERT LENGTH OK
; rung 50
LD 4582.01  ; BEARING INSERT LENGTH OK
ORNOT H356.09  ; Bearing insert having
AND 4582.00  ; OVERALL LENGTH OK
@AND T1552  ; CHECK TIME
OR 4582.02  ; LENGTH CHECK OK
LD H155.05  ; 10ST_STEP 05
OR H155.06  ; 10ST_STEP 06
OR H155.07  ; 10ST_STEP 07
OR 4591.04  ; Upper limit master check
OR 4591.08  ; Lower limit master check
ANDLD
OUT 4582.02  ; LENGTH CHECK OK
; rung 51
LDNOT 4582.01  ; BEARING INSERT LENGTH OK
AND H356.09  ; Bearing insert having
ORNOT 4582.00  ; OVERALL LENGTH OK
@AND T1552  ; CHECK TIME
OR 4582.03  ; LENGTH CHECK NG
LD H155.05  ; 10ST_STEP 05
OR H155.06  ; 10ST_STEP 06
OR H155.07  ; 10ST_STEP 07
OR 4591.04  ; Upper limit master check
OR 4591.08  ; Lower limit master check
ANDLD
LD H356.00  ; LENGTH WORKPIECE
AND 4581.10
ORLD
OUT 4582.03  ; LENGTH CHECK NG

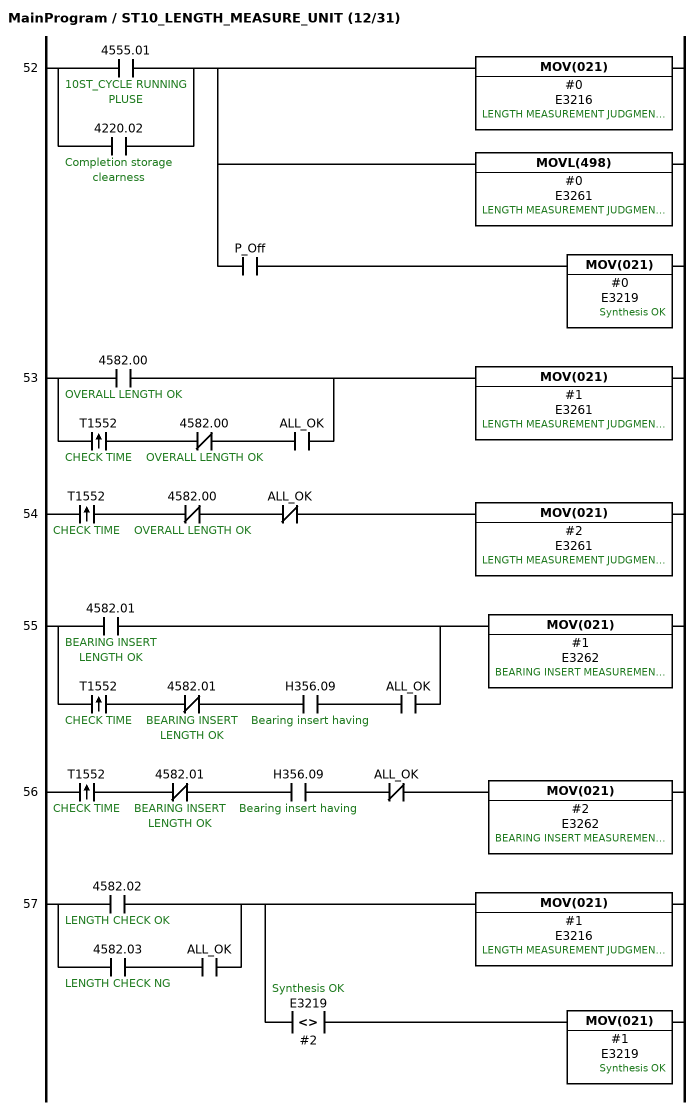
; rung 52
LD 4555.01  ; 10ST_CYCLE RUNNING PLUSE
OR 4220.02  ; Completion storage clearness
MOV(021) #0 E3216  ; LENGTH MEASUREMENT JUDGMENT RESULT (1:OK,2:NG)
MOVL(498) #0 E3261  ; LENGTH MEASUREMENT JUDGMENT RESULT (1:OK,2:NG)
AND P_Off
MOV(021) #0 E3219  ; Synthesis OK
; rung 53
LD 4582.00  ; OVERALL LENGTH OK
@LD T1552  ; CHECK TIME
ANDNOT 4582.00  ; OVERALL LENGTH OK
AND ALL_OK
ORLD
MOV(021) #1 E3261  ; LENGTH MEASUREMENT JUDGMENT RESULT (1:OK,2:NG)
; rung 54
@LD T1552  ; CHECK TIME
ANDNOT 4582.00  ; OVERALL LENGTH OK
ANDNOT ALL_OK
MOV(021) #2 E3261  ; LENGTH MEASUREMENT JUDGMENT RESULT (1:OK,2:NG)
; rung 55
LD 4582.01  ; BEARING INSERT LENGTH OK
@LD T1552  ; CHECK TIME
ANDNOT 4582.01  ; BEARING INSERT LENGTH OK
AND H356.09  ; Bearing insert having
AND ALL_OK
ORLD
MOV(021) #1 E3262  ; BEARING INSERT MEASUREMENT  JUDGMENT RESULT (1:OK,2:NG)
; rung 56
@LD T1552  ; CHECK TIME
ANDNOT 4582.01  ; BEARING INSERT LENGTH OK
AND H356.09  ; Bearing insert having
ANDNOT ALL_OK
MOV(021) #2 E3262  ; BEARING INSERT MEASUREMENT  JUDGMENT RESULT (1:OK,2:NG)
; rung 57
LD 4582.02  ; LENGTH CHECK OK
LD 4582.03  ; LENGTH CHECK NG
AND ALL_OK
ORLD
MOV(021) #1 E3216  ; LENGTH MEASUREMENT JUDGMENT RESULT (1:OK,2:NG)
AND<>(305) E3219 #2  ; Synthesis OK
MOV(021) #1 E3219  ; Synthesis OK

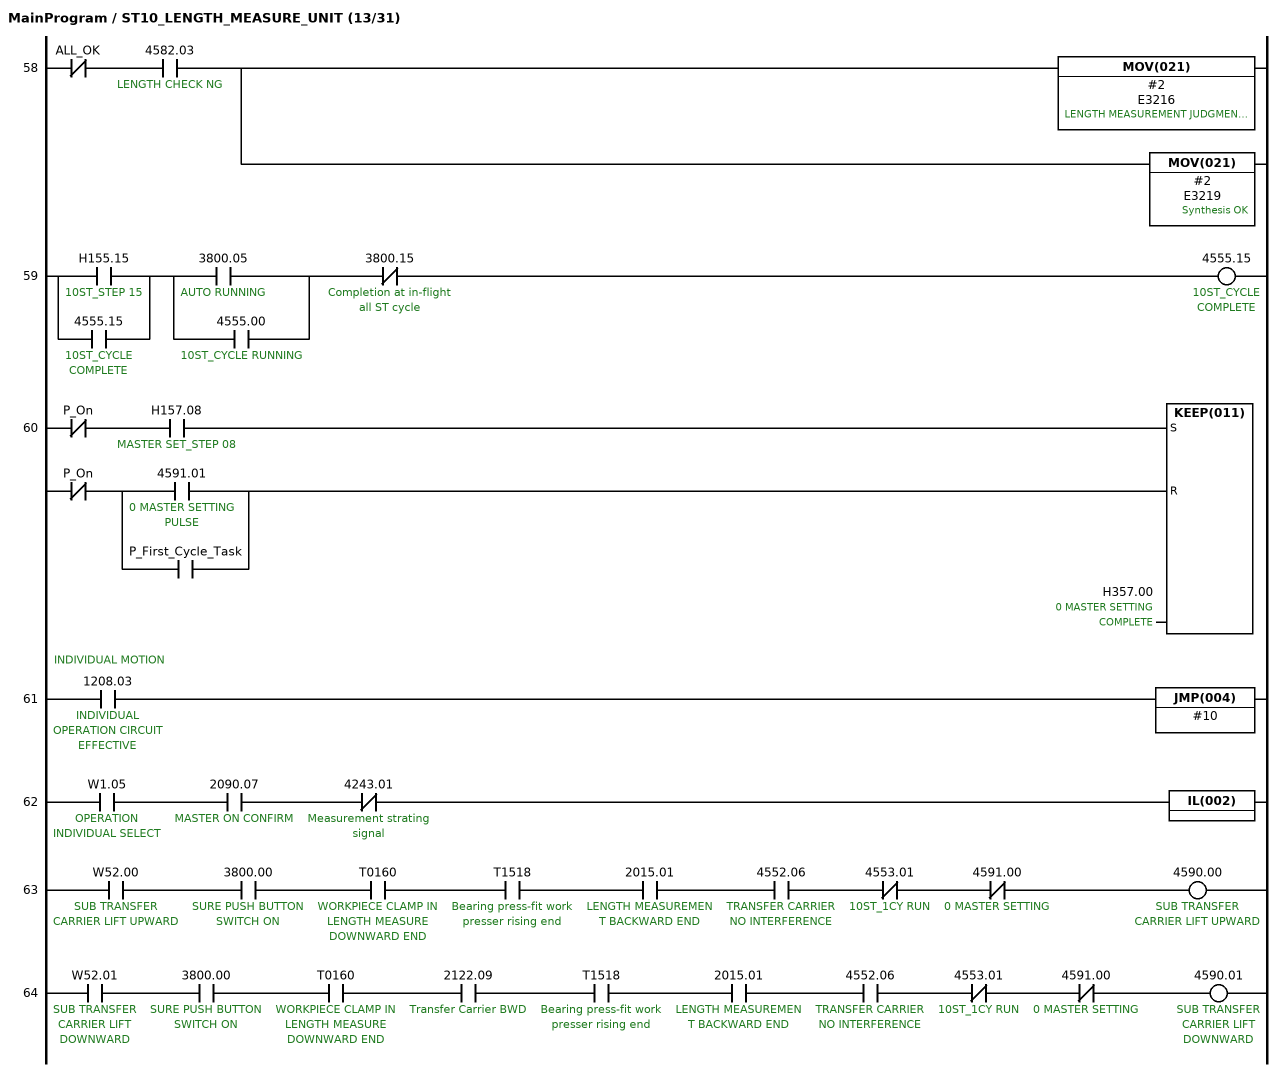
; rung 58
LDNOT ALL_OK
AND 4582.03  ; LENGTH CHECK NG
MOV(021) #2 E3216  ; LENGTH MEASUREMENT JUDGMENT RESULT (1:OK,2:NG)
MOV(021) #2 E3219  ; Synthesis OK
; rung 59
LD H155.15  ; 10ST_STEP 15
OR 4555.15  ; 10ST_CYCLE COMPLETE
LD 3800.05  ; AUTO RUNNING
OR 4555.00  ; 10ST_CYCLE RUNNING
ANDLD
ANDNOT 3800.15  ; Completion at in-flight all ST cycle
OUT 4555.15  ; 10ST_CYCLE COMPLETE
; rung 60
LDNOT P_On
AND H157.08  ; MASTER SET_STEP 08
LDNOT P_On
LD 4591.01  ; 0 MASTER SETTING PULSE
OR P_First_Cycle_Task
ANDLD
KEEP(011) H357.00  ; 0 MASTER SETTING COMPLETE
; rung 61: INDIVIDUAL MOTION
LD 1208.03  ; INDIVIDUAL OPERATION CIRCUIT EFFECTIVE
JMP(004) #10
; rung 62
LD W1.05  ; OPERATION INDIVIDUAL SELECT
AND 2090.07  ; MASTER ON CONFIRM
ANDNOT 4243.01  ; Measurement strating signal
IL(002)
; rung 63
LD W52.00  ; SUB TRANSFER CARRIER LIFT UPWARD
AND 3800.00  ; SURE PUSH BUTTON SWITCH ON
AND T0160  ; WORKPIECE CLAMP IN LENGTH MEASURE DOWNWARD END
AND T1518  ; Bearing press-fit work presser rising end
AND 2015.01  ; LENGTH MEASUREMENT BACKWARD END
AND 4552.06  ; TRANSFER CARRIER NO INTERFERENCE
ANDNOT 4553.01  ; 10ST_1CY RUN
ANDNOT 4591.00  ; 0 MASTER SETTING
OUT 4590.00  ; SUB TRANSFER CARRIER LIFT UPWARD
; rung 64
LD W52.01  ; SUB TRANSFER CARRIER LIFT DOWNWARD
AND 3800.00  ; SURE PUSH BUTTON SWITCH ON
AND T0160  ; WORKPIECE CLAMP IN LENGTH MEASURE DOWNWARD END
AND 2122.09  ; Transfer Carrier BWD
AND T1518  ; Bearing press-fit work presser rising end
AND 2015.01  ; LENGTH MEASUREMENT BACKWARD END
AND 4552.06  ; TRANSFER CARRIER NO INTERFERENCE
ANDNOT 4553.01  ; 10ST_1CY RUN
ANDNOT 4591.00  ; 0 MASTER SETTING
OUT 4590.01  ; SUB TRANSFER CARRIER LIFT DOWNWARD

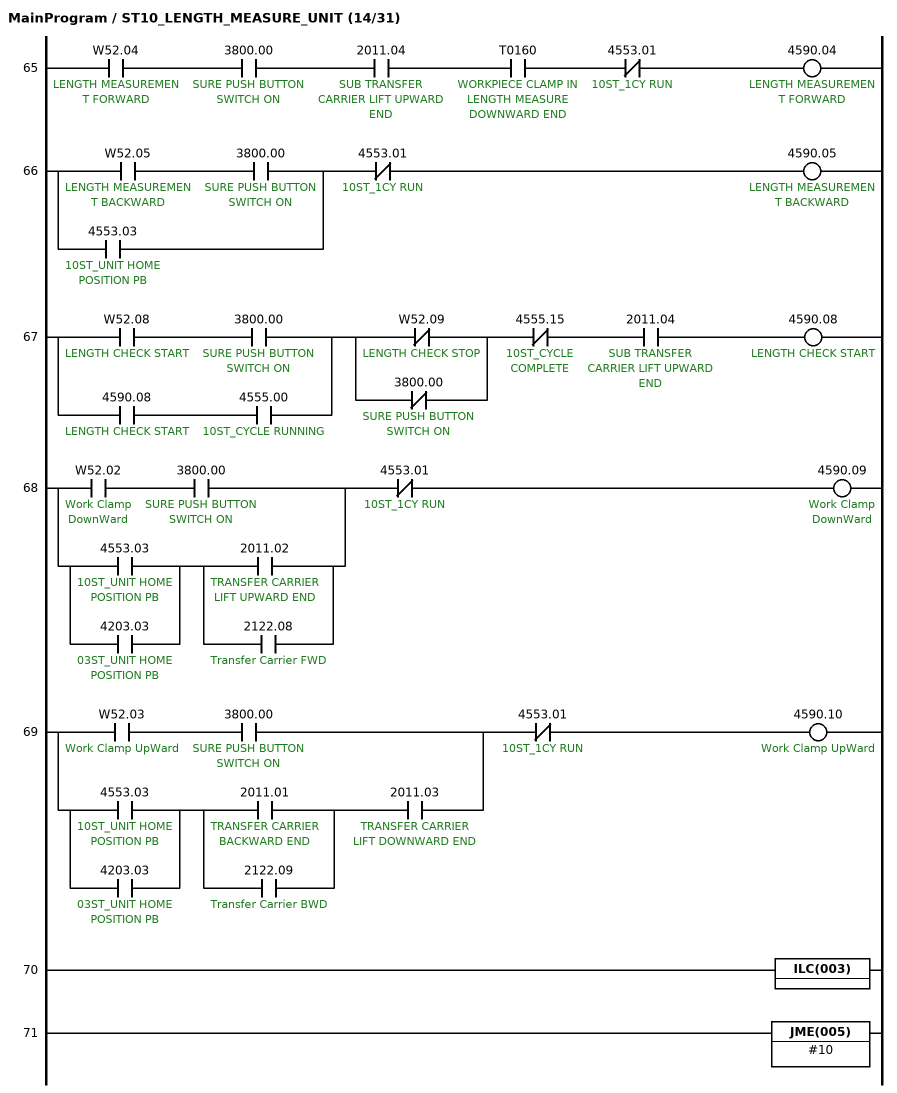
; rung 65
LD W52.04  ; LENGTH MEASUREMENT FORWARD
AND 3800.00  ; SURE PUSH BUTTON SWITCH ON
AND 2011.04  ; SUB TRANSFER CARRIER LIFT UPWARD END
AND T0160  ; WORKPIECE CLAMP IN LENGTH MEASURE DOWNWARD END
ANDNOT 4553.01  ; 10ST_1CY RUN
OUT 4590.04  ; LENGTH MEASUREMENT FORWARD
; rung 66
LD W52.05  ; LENGTH MEASUREMENT BACKWARD
AND 3800.00  ; SURE PUSH BUTTON SWITCH ON
OR 4553.03  ; 10ST_UNIT HOME POSITION PB
ANDNOT 4553.01  ; 10ST_1CY RUN
OUT 4590.05  ; LENGTH MEASUREMENT BACKWARD
; rung 67
LD W52.08  ; LENGTH CHECK START
AND 3800.00  ; SURE PUSH BUTTON SWITCH ON
LD 4590.08  ; LENGTH CHECK START
AND 4555.00  ; 10ST_CYCLE RUNNING
ORLD
LDNOT W52.09  ; LENGTH CHECK STOP
ORNOT 3800.00  ; SURE PUSH BUTTON SWITCH ON
ANDLD
ANDNOT 4555.15  ; 10ST_CYCLE COMPLETE
AND 2011.04  ; SUB TRANSFER CARRIER LIFT UPWARD END
OUT 4590.08  ; LENGTH CHECK START
; rung 68
LD W52.02  ; Work Clamp DownWard
AND 3800.00  ; SURE PUSH BUTTON SWITCH ON
LD 4553.03  ; 10ST_UNIT HOME POSITION PB
OR 4203.03  ; 03ST_UNIT HOME POSITION PB
LD 2011.02  ; TRANSFER CARRIER LIFT UPWARD END
OR 2122.08  ; Transfer Carrier FWD
ANDLD
ORLD
ANDNOT 4553.01  ; 10ST_1CY RUN
OUT 4590.09  ; Work Clamp DownWard
; rung 69
LD W52.03  ; Work Clamp UpWard
AND 3800.00  ; SURE PUSH BUTTON SWITCH ON
LD 4553.03  ; 10ST_UNIT HOME POSITION PB
OR 4203.03  ; 03ST_UNIT HOME POSITION PB
LD 2011.01  ; TRANSFER CARRIER BACKWARD END
OR 2122.09  ; Transfer Carrier BWD
ANDLD
AND 2011.03  ; TRANSFER CARRIER LIFT DOWNWARD END
ORLD
ANDNOT 4553.01  ; 10ST_1CY RUN
OUT 4590.10  ; Work Clamp UpWard
; rung 70
ILC(003)
; rung 71
JME(005) #10

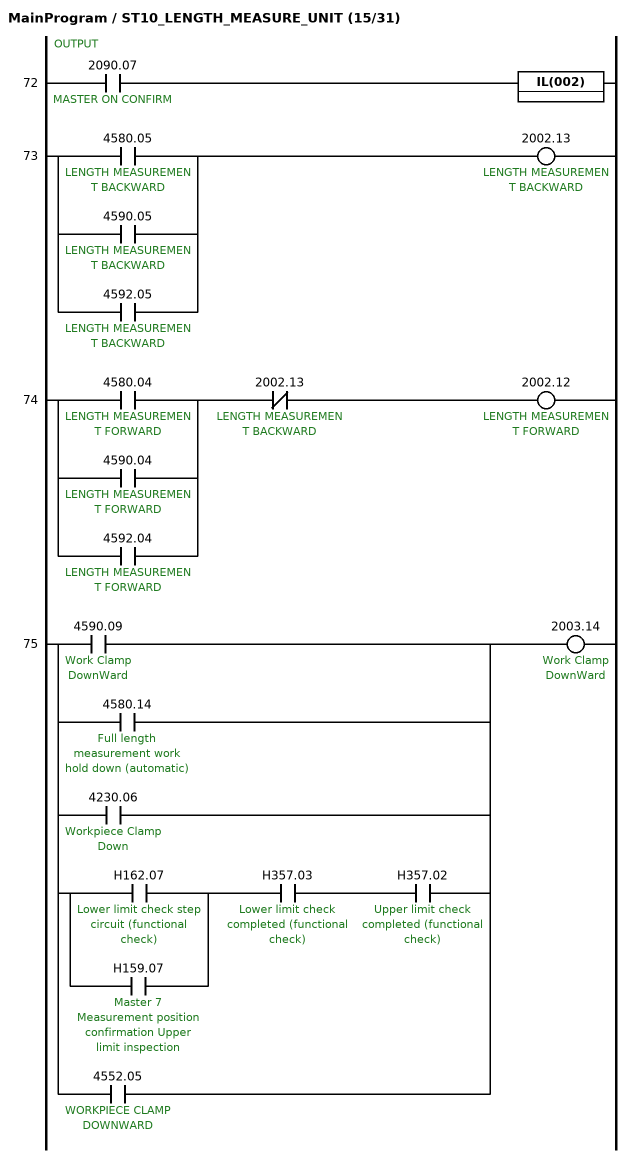
; rung 72: OUTPUT
LD 2090.07  ; MASTER ON CONFIRM
IL(002)
; rung 73
LD 4580.05  ; LENGTH MEASUREMENT BACKWARD
OR 4590.05  ; LENGTH MEASUREMENT BACKWARD
OR 4592.05  ; LENGTH MEASUREMENT BACKWARD
OUT 2002.13  ; LENGTH MEASUREMENT BACKWARD
; rung 74
LD 4580.04  ; LENGTH MEASUREMENT FORWARD
OR 4590.04  ; LENGTH MEASUREMENT FORWARD
OR 4592.04  ; LENGTH MEASUREMENT FORWARD
ANDNOT 2002.13  ; LENGTH MEASUREMENT BACKWARD
OUT 2002.12  ; LENGTH MEASUREMENT FORWARD
; rung 75
LD 4590.09  ; Work Clamp DownWard
OR 4580.14  ; Full length measurement work hold down (automatic)
OR 4230.06  ; Workpiece Clamp Down
LD H162.07  ; Lower limit check step circuit (functional check)
OR H159.07  ; Master 7 Measurement position confirmation Upper limit inspection
AND H357.03  ; Lower limit check completed (functional check)
AND H357.02  ; Upper limit check completed (functional check)
ORLD
OR 4552.05  ; WORKPIECE CLAMP DOWNWARD
OUT 2003.14  ; Work Clamp DownWard

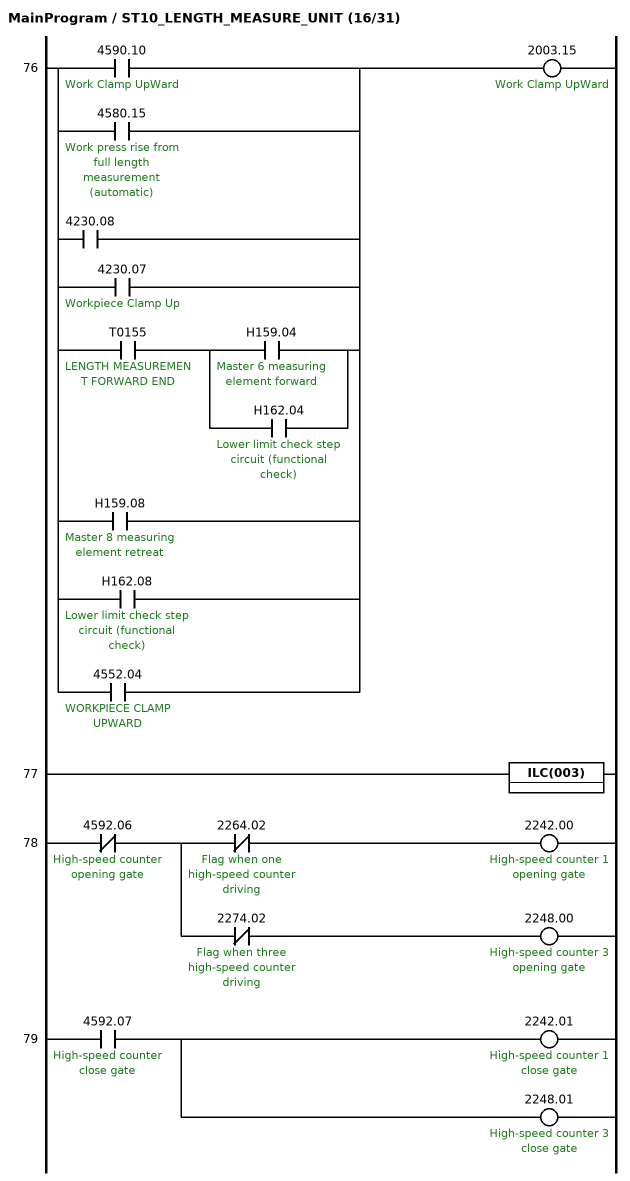
; rung 76
LD 4590.10  ; Work Clamp UpWard
OR 4580.15  ; Work press rise from full length measurement (automatic)
OR 4230.08
OR 4230.07  ; Workpiece Clamp Up
LD T0155  ; LENGTH MEASUREMENT FORWARD END
LD H159.04  ; Master 6 measuring element forward
OR H162.04  ; Lower limit check step circuit (functional check)
ANDLD
ORLD
OR H159.08  ; Master 8 measuring element retreat
OR H162.08  ; Lower limit check step circuit (functional check)
OR 4552.04  ; WORKPIECE CLAMP UPWARD
OUT 2003.15  ; Work Clamp UpWard
; rung 77
ILC(003)
; rung 78
LDNOT 4592.06  ; High-speed counter opening gate
OUT TR0
ANDNOT 2264.02  ; Flag when one high-speed counter driving
OUT 2242.00  ; High-speed counter 1 opening gate
LD TR0
ANDNOT 2274.02  ; Flag when three high-speed counter driving
OUT 2248.00  ; High-speed counter 3 opening gate
; rung 79
LD 4592.07  ; High-speed counter close gate
OUT 2242.01  ; High-speed counter 1 close gate
OUT 2248.01  ; High-speed counter 3 close gate

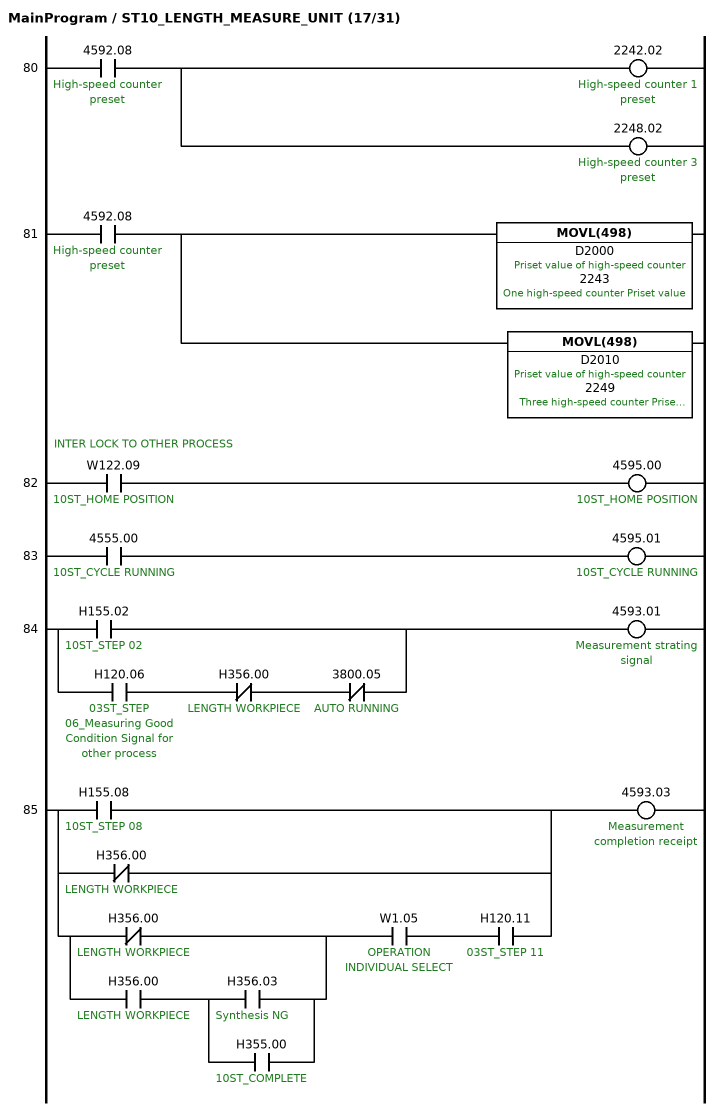
; rung 80
LD 4592.08  ; High-speed counter preset
OUT 2242.02  ; High-speed counter 1 preset
OUT 2248.02  ; High-speed counter 3 preset
; rung 81
LD 4592.08  ; High-speed counter preset
MOVL(498) D2000 2243  ; Priset value of high-speed counter, One high-speed counter Priset value
MOVL(498) D2010 2249  ; Priset value of high-speed counter, Three high-speed counter Priset value
; rung 82: INTER LOCK TO OTHER PROCESS
LD W122.09  ; 10ST_HOME POSITION
OUT 4595.00  ; 10ST_HOME POSITION
; rung 83
LD 4555.00  ; 10ST_CYCLE RUNNING
OUT 4595.01  ; 10ST_CYCLE RUNNING
; rung 84
LD H155.02  ; 10ST_STEP 02
LD H120.06  ; 03ST_STEP 06_Measuring Good Condition Signal for other process
ANDNOT H356.00  ; LENGTH WORKPIECE
ANDNOT 3800.05  ; AUTO RUNNING
ORLD
OUT 4593.01  ; Measurement strating signal
; rung 85
LD H155.08  ; 10ST_STEP 08
ORNOT H356.00  ; LENGTH WORKPIECE
LDNOT H356.00  ; LENGTH WORKPIECE
LD H356.00  ; LENGTH WORKPIECE
LD H356.03  ; Synthesis NG
OR H355.00  ; 10ST_COMPLETE
ANDLD
ORLD
AND W1.05  ; OPERATION INDIVIDUAL SELECT
AND H120.11  ; 03ST_STEP 11
ORLD
OUT 4593.03  ; Measurement completion receipt

